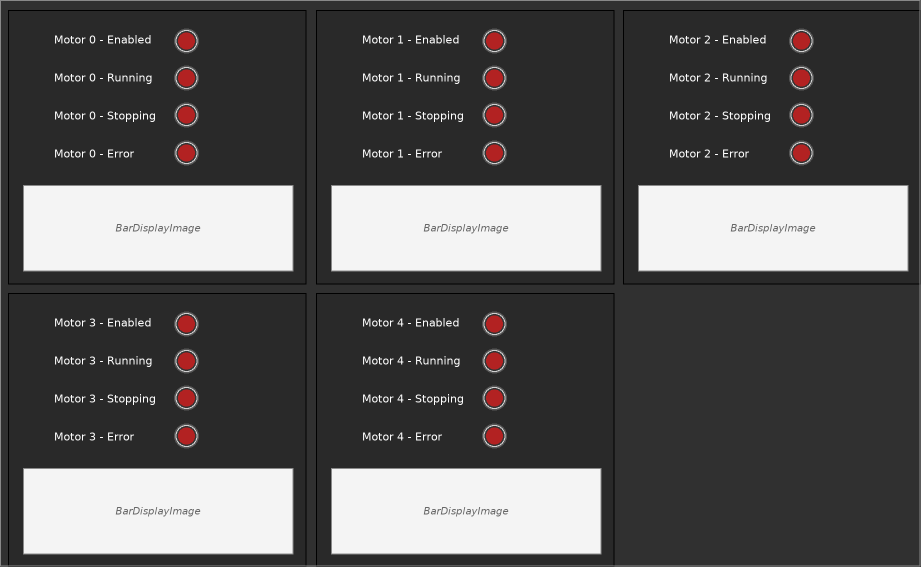
VISUALIZATION motor_status  // 921x567
    Rectangle (8,10 298x274)
    Label (51,25 150x30), "Motor 0 - Enabled"
    BarDisplayImage (23,185 270x86), value: MAIN.Motor[0].ref.NcToPlc.ActVelo, style: BarDisplayImage-Gray, scale format: %.1f, scale 0..2000
        p518627256: Motor 0 - Speed
    Lamp1 (172,26 29x30), variable: MAIN.Motor[0].fbPower.Status, style: Lamp-Lamp1-Red
    Label (51,63 150x30), "Motor 0 - Running"
    Label (51,101 150x30), "Motor 0 - Stopping"
    Label (51,139 150x30), "Motor 0 - Error"
    Lamp1 (172,63 29x30), variable: MAIN.Motor[0].ref.Status.Moving, style: Lamp-Lamp1-Red
    Lamp1 (172,100 29x30), variable: MAIN.Motor[0].ref.Status.Stopping, style: Lamp-Lamp1-Red
    Lamp1 (172,138 29x30), variable: MAIN.Motor[0].ref.Status.Error, style: Lamp-Lamp1-Red
    Rectangle (316,10 298x274)
    Label (359,25 150x30), "Motor 1 - Enabled"
    BarDisplayImage (331,185 270x86), value: MAIN.Motor[1].ref.NcToPlc.ActVelo, style: BarDisplayImage-Gray, scale format: %.1f, scale 0..2000
        p518627256: Motor 1 - Speed
    Lamp1 (480,26 29x30), variable: MAIN.Motor[1].fbPower.Status, style: Lamp-Lamp1-Red
    Label (359,63 150x30), "Motor 1 - Running"
    Label (359,101 150x30), "Motor 1 - Stopping"
    Label (359,139 150x30), "Motor 1 - Error"
    Lamp1 (480,63 29x30), variable: MAIN.Motor[1].ref.Status.Moving, style: Lamp-Lamp1-Red
    Lamp1 (480,100 29x30), variable: MAIN.Motor[1].ref.Status.Stopping, style: Lamp-Lamp1-Red
    Lamp1 (480,138 29x30), variable: MAIN.Motor[1].ref.Status.Error, style: Lamp-Lamp1-Red
    Rectangle (623,10 298x274)
    Label (666,25 150x30), "Motor 2 - Enabled"
    BarDisplayImage (638,185 270x86), value: MAIN.Motor[2].ref.NcToPlc.ActVelo, style: BarDisplayImage-Gray, scale format: %.1f, scale 0..2000
        p518627256: Motor 2 - Speed
    Lamp1 (787,26 29x30), variable: MAIN.Motor[2].fbPower.Status, style: Lamp-Lamp1-Red
    Label (666,63 150x30), "Motor 2 - Running"
    Label (666,101 150x30), "Motor 2 - Stopping"
    Label (666,139 150x30), "Motor 2 - Error"
    Lamp1 (787,63 29x30), variable: MAIN.Motor[2].ref.Status.Moving, style: Lamp-Lamp1-Red
    Lamp1 (787,100 29x30), variable: MAIN.Motor[2].ref.Status.Stopping, style: Lamp-Lamp1-Red
    Lamp1 (787,138 29x30), variable: MAIN.Motor[2].ref.Status.Error, style: Lamp-Lamp1-Red
    Rectangle (8,293 298x274)
    Label (51,308 150x30), "Motor 3 - Enabled"
    BarDisplayImage (23,468 270x86), value: MAIN.Motor[3].ref.NcToPlc.ActVelo, style: BarDisplayImage-Gray, scale format: %.1f, scale 0..2000
        p518627256: Motor 3 - Speed
    Lamp1 (172,309 29x30), variable: MAIN.Motor[3].fbPower.Status, style: Lamp-Lamp1-Red
    Label (51,346 150x30), "Motor 3 - Running"
    Label (51,384 150x30), "Motor 3 - Stopping"
    Label (51,422 150x30), "Motor 3 - Error"
    Lamp1 (172,346 29x30), variable: MAIN.Motor[3].ref.Status.Moving, style: Lamp-Lamp1-Red
    Lamp1 (172,383 29x30), variable: MAIN.Motor[3].ref.Status.Stopping, style: Lamp-Lamp1-Red
    Lamp1 (172,421 29x30), variable: MAIN.Motor[3].ref.Status.Error, style: Lamp-Lamp1-Red
    Rectangle (316,293 298x274)
    Label (359,308 150x30), "Motor 4 - Enabled"
    BarDisplayImage (331,468 270x86), value: MAIN.Motor[4].ref.NcToPlc.ActVelo, style: BarDisplayImage-Gray, scale format: %.1f, scale 0..2000
        p518627256: Motor 4 - Speed
    Lamp1 (480,309 29x30), variable: MAIN.Motor[4].fbPower.Status, style: Lamp-Lamp1-Red
    Label (359,346 150x30), "Motor 4 - Running"
    Label (359,384 150x30), "Motor 4 - Stopping"
    Label (359,422 150x30), "Motor 4 - Error"
    Lamp1 (480,346 29x30), variable: MAIN.Motor[4].ref.Status.Moving, style: Lamp-Lamp1-Red
    Lamp1 (480,383 29x30), variable: MAIN.Motor[4].ref.Status.Stopping, style: Lamp-Lamp1-Red
    Lamp1 (480,421 29x30), variable: MAIN.Motor[4].ref.Status.Error, style: Lamp-Lamp1-Red
END_VISUALIZATION

(* stored: Version 1.1.0.1, ProductVersion 3.1.4024.11
   Visu motor_status: Id {9bfc1aee-9021-4fb8-9ba1-0af391d43a27} *)
